FUNCTION_BLOCK FB_OPCUA_ClientConnection IMPLEMENTS I_OPCUA_ClientConnection
VAR_INPUT
END_VAR
VAR_OUTPUT
	connectionHdl : DWORD;
	nNamespaceIndex			: UINT;
	connectDone : BOOL;
	disconnectDone : BOOL;
	error : BOOL;
END_VAR
VAR
	nameSpaceLocationIdentifierEx : STRING(MAX_STRING_LENGTH); 
	NamespaceUriEx : STRING(MAX_STRING_LENGTH); 
	_iOPCUA_Connect			: I_OPCUA_COnnect;
	SessionConnectInfoEx	: ST_UASessionConnectInfo;
	_iOPCUA_GetNameSpaceIndex 	: I_OPCUA_GetNameSpaceIndex;
	
	(* Declarations for disconnect*)
	_iOPCUA_Disconnect		: I_OPCUA_Disconnect;
	
	(* Other declarations *) 
	writeStep : INT;
	errorID : DWORD;	
	executing : BOOL;
	firstTimeWrite : BOOL;
	serverURLex: STRING(MAX_STRING_LENGTH);
	connectStep: INT;
	disconnectStep: INT;
	connectBusy: BOOL;
	connectError: BOOL;
	getNameSpaceIndexBusy: BOOL;
	getNameSpaceIndexError: BOOL;
	disconnectBusy: BOOL;
	disconnectError: BOOL;
	getNameSpaceErrorID: DWORD;
	connectErrorID: DWORD;
END_VAR

{warning 'add method implementation '}
METHOD connect : BOOL
VAR_INPUT
	(* server address *)
	serverUrl	: STRING(MAX_STRING_LENGTH);
	(* namespace uri*)
	namespaceUri	: STRING(MAX_STRING_LENGTH);
	(* Location of data in namespace *)
	nameSpaceLocationIdentifier	: STRING(MAX_STRING_LENGTH);
	(* Session connect info struct *)
	sessionConnectInfo	: ST_UASessionConnectInfo;
END_VAR


CASE connectStep OF
	0:
		error := FALSE;
		connectDone := FALSE;
		disconnectStep := 0;
		nameSpaceUriEx := namespaceUri;
		sessionConnectInfoEx := SessionConnectInfo;
		serverURlex := serverUrl;
		nameSpaceLocationIdentifierEx := nameSpaceLocationIdentifier;
		SessionConnectInfoEx.sApplicationName := 'asddddd';
		_iOPCUA_Connect.start(
			Execute				:= TRUE,
			ServerURL			:= serverURLex,
			SessionConnectInfo  := SessionConnectInfoEx,
			Timeout				:= T#2M,
			ConnectionHdl		=> ConnectionHdl,
			busy				=> connectBusy,
			error				=> connectError,
			errorID				=> connectErrorID
		);
		IF NOT connectBusy THEN
			_iOPCUA_Connect.start(Execute := FALSE,
								ServerURL			:= serverURLex,
								SessionConnectInfo  := SessionConnectInfoEx,
								Timeout				:= T#2M,
								ConnectionHdl		=> ConnectionHdl
								);
	
			IF NOT connectError THEN
				(* session open *)
				connectStep :=connectStep + 1;
			ELSE
				Error			:= TRUE;
				ErrorID		:= connectErrorID;
				ConnectionHdl	:= 0;
				writeStep		:= 0; (* idle *)
			END_IF
		END_IF
	1:
		_iOPCUA_GetNameSpaceIndex.start(
										Execute			:= TRUE,
										ConnectionHdl	:= ConnectionHdl,
										NamespaceUri	:= NamespaceUriEx,
										TimeOut 		:= T#5S,
										NamespaceIndex	=> nNamespaceIndex,
										busy			=> getNameSpaceIndexBusy,
										error			=> getNameSpaceIndexError,
										errorID			=> getNameSpaceErrorID
										);
	
	
		IF NOT getNameSpaceIndexBusy THEN
			_iOPCUA_GetNameSpaceIndex.start(Execute := FALSE,
											ConnectionHdl	:= ConnectionHdl,
											NamespaceUri	:= NamespaceUriEx,
											TimeOut 		:= T#5S,
											NamespaceIndex	=> nNamespaceIndex,
											);
			IF NOT getNameSpaceIndexError THEN
				(* session closed *)
				connectDone := TRUE;
				connectStep 	:= 0; (* idle *)
			ELSE
				Error		:= TRUE;
				ErrorID	:= getNameSpaceErrorID;
				connectStep := 0;
				// CLEANUP?writeStep 		:= 5; (* idle *)
			END_IF
		END_IF	
END_CASE
END_METHOD

{warning 'add method implementation '}
METHOD disconnect : BOOL

VAR
	Execute: INT;
	disconnectErrorID: DWORD;
END_VAR
CASE disconnectStep OF
	0:	(* close session *)
		error := FALSE;
		disconnectDone := FALSE;
		connectStep := 0;
		_iOPCUA_Disconnect.start(
							Execute			:= TRUE,
							ConnectionHdl	:= connectionHdl,
							timeOut			:= T#5S,
							busy			=> disconnectBusy,
							error			=> disconnectError,
							errorID			=> disconnectErrorID
						);
	
		IF NOT disconnectBusy THEN
			_iOPCUA_Disconnect.start(Execute := FALSE,
									ConnectionHdl	:= connectionHdl,
									timeOut			:= T#5S
									);
			//Busy := FALSE;
			IF NOT disconnectError THEN
				(* session closed *)
				firstTimeWrite := TRUE;
	//			firstTimeWrite := FALSE;
				Executing := FALSE;
//				clientVariablePrev := clientVariable.pValue^;
				disconnectStep 		:= 0; (* idle *)
				IF NOT error THEN 
					disconnectDone := TRUE;
					disconnectStep := 0;
				END_IF
			ELSE
				error			:= TRUE;
				//lastErrorStep := 6;
				errorID		:= disconnectErrorID;
				//writeStep 			:= 0; (* idle *)
				connectionHdl	:= 0;
			END_IF
		END_IF	
END_CASE
END_METHOD

METHOD FB_init : BOOL
VAR_INPUT
	bInitRetains : BOOL; // if TRUE, the retain variables are initialized (warm start / cold start)
	bInCopyCode : BOOL;  // if TRUE, the instance afterwards gets moved into the copy code (online change)
	iOPCUAconnect : I_OPCUA_Connect;
	iOPCUAdisconnect : I_OPCUA_Disconnect;
	iOPCUAgetNameSpaceIndex : I_OPCUA_GetNameSpaceIndex; 
END_VAR
_iOPCUA_Connect := iOPCUAconnect;
_iOPCUA_Disconnect := iOPCUAdisconnect;
_iOPCUA_GetNameSpaceIndex := iOPCUAgetNameSpaceIndex;
END_METHOD

END_FUNCTION_BLOCK

(* stored: Version 1.1.0.1, ProductVersion 3.1.4024.9
   POU FB_OPCUA_ClientConnection: Id {d4ee0b34-a2a9-445d-aa96-86e0d20319fc}, SpecialFunc None
   Method connect: Id {1316d943-629f-4de0-857d-49fc71159adf}
   Method disconnect: Id {985ae0bf-e099-417e-89f9-f09db7a9b7a9}
   Method FB_init: Id {c91b2b38-559f-4490-bb3d-4d027253fec9} *)
